TYPE
    Data EXTENDS TcoData.Entity :
    STRUCT
        sampleData : SampleDataStructure;
    END_STRUCT
END_TYPE

(* stored: Version 1.1.0.1, ProductVersion 3.1.4024.9
   DUT Data: Id {db6560ed-fb2a-0049-1f52-f29952b65ec0} *)
